(* PLC project new_mac, Dassault Systèmes ControlBuild 2024x Refresh1 *)
(* stored: creationDateTime 2024-04-11T13:53:43-01:00 *)

PROGRAM robot6axis_ctrled.new_mac

(* FBD diagram, written out as Structured Text *)
END_PROGRAM
